INTERFACE I_ImageSerializer

METHOD PUBLIC ConnectTo
VAR_INPUT
	ImageSerializer : I_ImageSerializer;
END_VAR
END_METHOD

METHOD PUBLIC GetTotalSerializablePixelCount : UDINT
VAR_INPUT
END_VAR
END_METHOD

PROPERTY PUBLIC PixelCount : UDINT
GET
END_GET
END_PROPERTY

METHOD PUBLIC TryGetPixel : BOOL
VAR_INPUT
	PixelIndex : UDINT;
	Reader : I_PixelReader;
END_VAR
END_METHOD

METHOD PUBLIC UpdateImage
VAR_INPUT
	Source : ITcVnImage;
END_VAR
END_METHOD

END_INTERFACE

(* stored: Version 1.1.0.1
   Itf I_ImageSerializer: Id {cb305bac-5870-4b0c-a366-7d8a0d1281e6}
   Method ConnectTo: Id {ed84f8cb-c203-4f0b-bccd-097e6a749da6}
   Method GetTotalSerializablePixelCount: Id {5446371e-1f85-47a3-bbf1-b3ce25dfac0f}
   Property PixelCount: Id {40306301-2bbc-4248-a8d7-f5470f3fcfbf}
   Get Get: Id {0ec63ad1-f9d8-41dc-a7cd-de28431dba62}
   Method TryGetPixel: Id {f158a363-3806-4123-b656-8fdfacffcd87}
   Method UpdateImage: Id {5435dbba-a720-415d-a50a-5887d020598a} *)
